// TIA Portal project "s71500pidwebsever" (V16)

(* hardware
DEVICE "S71500/ET200MP station_1"  S7-1500 station
   slot 0: "Rail_0"  Rack  6ES7 590-1***0-0AA0
   slot 1: "PLC_1"  CPU 1512C-1 PN  6ES7 512-1CK01-0AB0  V2.8
      slot 3: "CPU display_1"  6ES7591-1AA00-0AA0
      slot 32768: "PROFINET interface_1"  X1
         slot 32769: "Port_1"  X1 P1
         slot 32770: "Port_2"  X1 P2
      slot 34817: "Virtual CP interface port_1"  Virtual CP interface port  Virtual CP interface port
*)

// ===== PLC "PLC_1"  CPU 1512C-1 PN =====

VAR_GLOBAL   // PLC tag table "Default tag table"
   "System_Byte" AT %MB1 : Byte;
   "FirstScan" AT %M1.0 : Bool;
   "DiagStatusUpdate" AT %M1.1 : Bool;
   "AlwaysTRUE" AT %M1.2 : Bool;
   "AlwaysFALSE" AT %M1.3 : Bool;
   "analog" AT %IW64 : Word;
   "start_system" AT %M0.0 : Bool;
   "Fan" AT %Q0.1 : Bool;
   "ON" AT %M0.1 : Bool;
   "OFF" AT %M0.2 : Bool;
   "Tag_1" AT %MW30 : Int;
   "Tag_2" AT %MW10 : Int;
   "Tag_3" AT %M2.1 : Bool;
   "Tag_4" AT %M2.2 : Bool;
   "STOP" AT %M0.3 : Bool;
END_VAR

DATA_BLOCK "Web_Comm"   // DB1
{ S7_Optimized_Access := 'FALSE' }
VERSION : 0.1
   VAR
      analog_in : Int;
      nhiet_do : Real;
      setpoint : Real;
      start : Bool;
      stop : Bool;
      trang_thai : Bool;
   END_VAR
BEGIN
END_DATA_BLOCK

FUNCTION "Analog_input" : Void   // FC1, LAD
{ S7_Optimized_Access := 'TRUE' }
VERSION : 0.1
   VAR_INPUT
      "analog-in" : Int;
      min1 : Int;
      max1 : Int;
      min2 : Real;
      max2 : Real;
   END_VAR
   VAR_OUTPUT
      "nhiet-do" : Real;
   END_VAR
   VAR_TEMP
      "temp-real" : Real;
   END_VAR
BEGIN

REGION Network 1
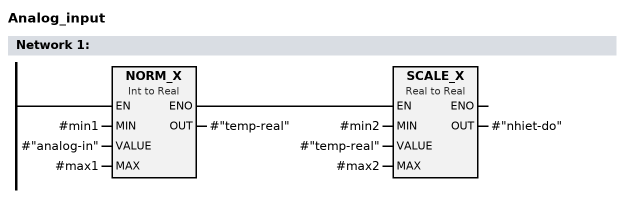
   RUNG wire#powerrail
      { S7_Templates := "[SrcType := Int, DestType := Real]" } Normalize(min := #min1, value := #"analog-in", max := #max1, out => #"temp-real")
      { S7_Templates := "[SrcType := Real, DestType := Real]" } Scale(min := #min2, value := #"temp-real", max := #max2, out => #"nhiet-do")
   END_RUNG
   // the same network as SCL:
   #"temp-real" := NORM_X(MIN := #min1, VALUE := #"analog-in", MAX := #max1);
   #"nhiet-do" := SCALE_X(MIN := #min2, VALUE := #"temp-real", MAX := #max2);
END_REGION
END_FUNCTION

ORGANIZATION_BLOCK "Main"   // OB1, LAD, ProgramCycle
TITLE = "Main Program Sweep (Cycle)"
{ S7_Optimized_Access := 'TRUE' }
VERSION : 0.1
   VAR_INPUT
      Initial_Call : Bool;   // Initial call of this OB
      Remanence : Bool;   // =True, if remanent data are available
   END_VAR
   VAR_TEMP   // added for the SCL form of the ladder/FBD networks
      _w1 : Bool;
   END_VAR
BEGIN

REGION Network 1
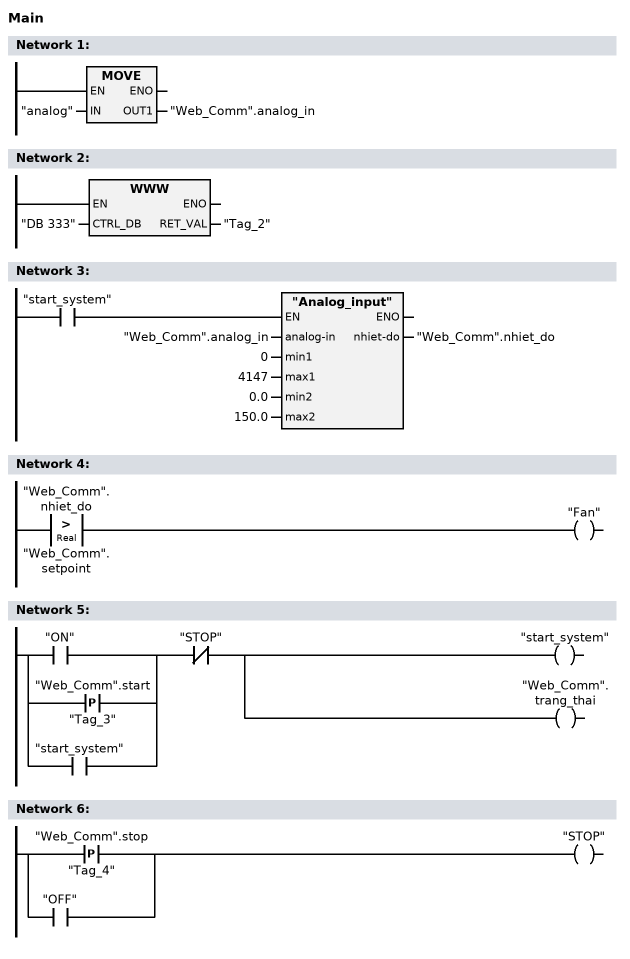
   RUNG wire#powerrail
      Move(in := "analog", out1 => "Web_Comm".analog_in)
   END_RUNG
   // the same network as SCL:
   "Web_Comm".analog_in := "analog";
END_REGION

REGION Network 2
   "Tag_2" := WWW(CTRL_DB := "DB 333");
END_REGION

REGION Network 3
   RUNG wire#powerrail
      Contact( "start_system" )
      "Analog_input"("analog-in" := "Web_Comm".analog_in, min1 := 0, max1 := 4147, min2 := 0.0, max2 := 150.0, "nhiet-do" => "Web_Comm".nhiet_do)
   END_RUNG
   // the same network as SCL:
   IF "start_system" THEN
       "Analog_input"("analog-in" := "Web_Comm".analog_in,
                      min1 := 0,
                      max1 := 4147,
                      min2 := 0.0,
                      max2 := 150.0,
                      "nhiet-do" => "Web_Comm".nhiet_do);
   END_IF;
END_REGION

REGION Network 4
   RUNG wire#powerrail
      { S7_Templates := "SrcType := Real" } GT_Contact(in1 := "Web_Comm".nhiet_do, in2 := "Web_Comm".setpoint)
      Coil( "Fan" )
   END_RUNG
   // the same network as SCL:
   "Fan" := "Web_Comm".nhiet_do > "Web_Comm".setpoint;
END_REGION

REGION Network 5
   RUNG wire#powerrail
      Contact( "ON" )
      wire#w1
      I_Contact( "STOP" )
      wire#w2
      Coil( "start_system" )
   END_RUNG
   RUNG wire#powerrail
      P_Contact(operand := "Web_Comm".start, bit := "Tag_3")
   END_RUNG wire#w1
   RUNG wire#powerrail
      Contact( "start_system" )
   END_RUNG wire#w1
   RUNG wire#w2
      Coil( "Web_Comm".trang_thai )
   END_RUNG
   // the same network as SCL:
   #_w1 := "Web_Comm".start AND NOT "Tag_3";   // rising edge of "Web_Comm".start
   "Tag_3" := "Web_Comm".start;
   "start_system" := ("ON" OR #_w1 OR "start_system") AND NOT "STOP";
   "Web_Comm".trang_thai := "start_system";
END_REGION

REGION Network 6
   RUNG wire#powerrail
      P_Contact(operand := "Web_Comm".stop, bit := "Tag_4")
      wire#w1
      Coil( "STOP" )
   END_RUNG
   RUNG wire#powerrail
      Contact( "OFF" )
   END_RUNG wire#w1
   // the same network as SCL:
   #_w1 := "Web_Comm".stop AND NOT "Tag_4";   // rising edge of "Web_Comm".stop
   "Tag_4" := "Web_Comm".stop;
   "STOP" := #_w1 OR "OFF";
END_REGION
END_ORGANIZATION_BLOCK

ORGANIZATION_BLOCK "Cyclic interrupt"   // OB30, LAD, CyclicInterrupt
{ S7_Optimized_Access := 'TRUE' }
VERSION : 0.1
   VAR_INPUT
      Initial_Call : Bool;   // Initial call of this OB
      Event_Count : Int;   // Events discarded
   END_VAR
BEGIN

REGION Network 1
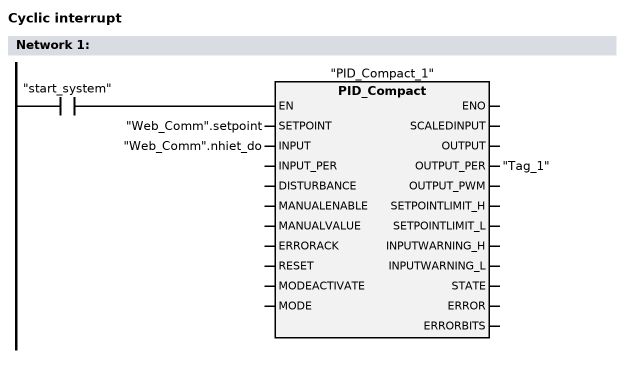
   IF "start_system" THEN
       "PID_Compact_1"(Setpoint := "Web_Comm".setpoint, Input := "Web_Comm".nhiet_do, Output_PER => "Tag_1");   // PID_Compact
   END_IF;
END_REGION
END_ORGANIZATION_BLOCK